(* IEC 61131-3 sources: windowtracking/src/lib/Windows, 3 files *)

(* ---- ITransportWindow.st ---- *)
USING Simatic.Ax.WindowTracking.Exits;
USING Simatic.Ax.SimpleControlModules;

NAMESPACE Simatic.Ax.WindowTracking
    INTERFACE ITransportWindow

        // METHOD GetTriggerPointCount : UINT
        // END_METHOD

        // METHOD GetTriggerPoint : ITriggerPoint
        //     VAR_INPUT
        //         Id : UINT;
        //     END_VAR
        // END_METHOD

        METHOD Reset
        END_METHOD

        METHOD CalcPosition
            VAR_INPUT
                enc : IEncoder;
            END_VAR
        END_METHOD

        METHOD GetPosition : DINT
        END_METHOD

    END_INTERFACE
END_NAMESPACE

(* ---- TransportWindow.st ---- *)
USING Simatic.Ax.SimpleControlModules;
USING Simatic.Ax.SimpleControlModules;
USING Simatic.Ax.WindowTracking.Exits;

NAMESPACE Simatic.Ax.WindowTracking

    CLASS TransportWindow IMPLEMENTS ITransportWindow
        VAR PUBLIC
        END_VAR
        VAR PROTECTED
            _actualPos : DINT;
            _lastPos : DINT;
        END_VAR

        METHOD PUBLIC CalcPosition
            VAR_INPUT
                enc : IEncoder;
            END_VAR
            VAR_TEMP
                _newPos : DINT;
                _difference : DINT;
            END_VAR
            _newPos := enc.GetValue();
            _difference := (_newPos - _lastPos) MOD enc.GetModulo();
            _actualPos := _actualPos + _difference;
        END_METHOD

        // METHOD PUBLIC CheckPos
        //     IF (Destination1 <> NULL) THEN
        //         Destination1.Check(THIS);
        //     END_IF;
        //     SortDecission.Check(THIS);
        // END_METHOD

        // METHOD PUBLIC GetTriggerPointCount : UINT
        //     IF (Destination1 <> NULL) THEN
        //         GetTriggerPointCount := UINT#1;
        //     ELSE
        //         GetTriggerPointCount := UINT#0;
        //     END_IF;
        // END_METHOD

        // METHOD PUBLIC GetTriggerPoint : ITriggerPoint
        //     VAR_INPUT
        //         Id : UINT;
        //     END_VAR
        //     IF (ID <> UINT#1) THEN
        //         GetTriggerPoint := NULL;
        //         RETURN;
        //     END_IF;

        //     IF (THIS.GetTriggerPointCount() = UINT#1) THEN
        //         GetTriggerPoint := Destination1;
        //         RETURN;
        //     END_IF;

        //     GetTriggerPoint := NULL;

        // END_METHOD

        METHOD PUBLIC GetExit : IExit
            ;
        END_METHOD

        METHOD PUBLIC Reset
            // Destination1 := NULL;
            _actualPos := 0;
            _lastPos := 0;
        END_METHOD
END_CLASS
END_NAMESPACE

(* ---- TransportWindows.st ---- *)
USING Simatic.Ax.SimpleControlModules;

NAMESPACE Simatic.Ax.WindowTracking
    CLASS TransportWindows
        VAR PUBLIC
            Encoder : IEncoder;
        END_VAR
        VAR PROTECTED
            _tranportWindowList : ARRAY[UINT#0..BUF_SIZE - UINT#1] OF ITransportWindow;
            _tranportWindowListStorage : ARRAY[UINT#0..BUF_SIZE - UINT#1] OF TransportWindow;
            _count : UINT;
            _head : UINT;
            _tail : UINT;
        END_VAR

        VAR CONSTANT
            BUF_SIZE : UINT := UINT#100;
        END_VAR

        METHOD PUBLIC Create
            _tranportWindowList[_head] := _tranportWindowListStorage[_head];
            _head := _head + UINT#1;
            _head := _head MOD BUF_SIZE;
        END_METHOD

        METHOD PUBLIC Remove
            IF (_tranportWindowList[_tail] <> NULL) THEN
                _tranportWindowListStorage[_tail].Reset();
                _tranportWindowList[_tail] := NULL;
                _tail := _tail + UINT#1;
                _tail := _tail MOD BUF_SIZE;
            END_IF;
        END_METHOD

        METHOD PUBLIC GetHead : UINT
            GetHead := _head;
        END_METHOD

        METHOD PUBLIC GetTail : UINT
            GetTail := _tail;
        END_METHOD

        METHOD PUBLIC GetWindow : ITransportWindow
             VAR_INPUT
                 id : UINT;
             END_VAR
             GetWindow := _tranportWindowListStorage[id];
        END_METHOD

        METHOD PUBLIC Count : UINT
            Count := ((_head - _tail) + BUF_SIZE) MOD BUF_SIZE;
        END_METHOD

        METHOD PUBLIC Evaluate
            VAR_TEMP
                i : UINT;
                o : ITransportWindow;
            END_VAR
            FOR i := UINT#0 TO THIS.Count() - UINT#1 DO
                o := _tranportWindowList[(_tail + i) MOD BUF_SIZE];
                IF (o <> NULL) THEN
                    o.CalcPosition(enc := Encoder);
                END_IF;
            END_FOR;
        END_METHOD
    END_CLASS
END_NAMESPACE
